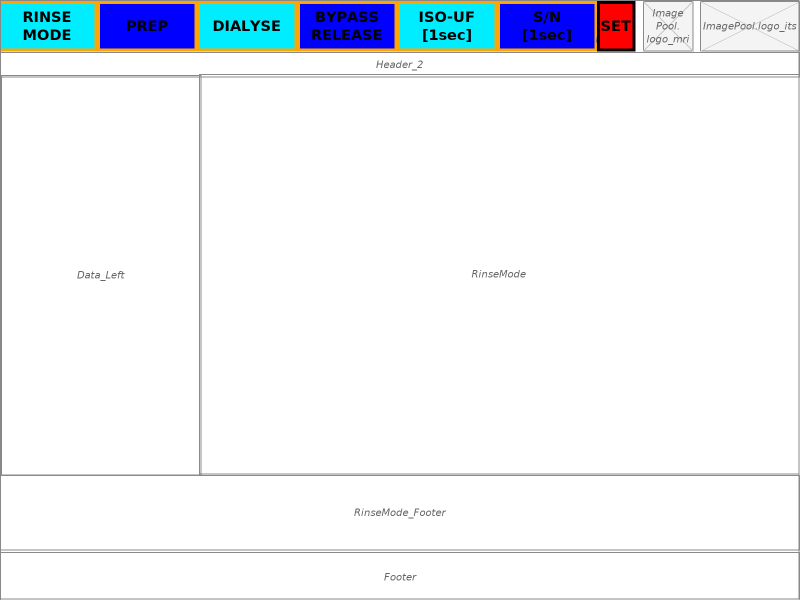
VISUALIZATION MainScreen  // 800x600
    Frame (0,52 800x25)
        shows Header_2()
    Frame (0,552 800x50)
        shows Footer()
    Frame (1,75 200x400)
        shows Data_Left()
    Frame (0,475 800x75)
        shows RinseMode_Footer()
    Rectangle (-3,1 100x50), "RINSE MODE"
        OnMouseClick: FrameSelectionChange Selection=SelectedFrame=2b0ef998-403b-4e78-a897-9d833b853fee, GlobSel=AssignType=Directly, SelType=Locally
    Rectangle (97,1 100x50), "PREP"
    Rectangle (197,1 100x50), "DIALYSE"
    Rectangle (297,1 100x50), "BYPASS RELEASE", tooltip "BY PAS"
    Rectangle (397,1 100x50), "ISO-UF [1sec]"
    Rectangle (497,1 100x50), "S/N [1sec]"
    Image (597,1 25x50), image: ImagePool.logo_its
    Image (643,1 50x50), image: ImagePool.logo_mri
    Rectangle (597,1 38x50), "SET"
        OnMouseClick: FrameSelectionChange Selection=SelectedFrame=2b0ef998-403b-4e78-a897-9d833b853fee, Selection=1, GlobSel=AssignType=Directly, SelType=Locally
    Image (700,1 100x50), image: ImagePool.logo_its
    Frame (199,74 600x400)
        shows RinseMode()
        shows Set()
END_VISUALIZATION

(* stored: Version 1.1.0.1, ProductVersion 3.1.4024.12
   Visu MainScreen: Id {6b497169-f106-4880-a797-d63f02820d0b} *)
